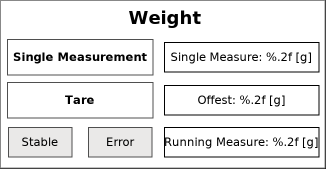
VISUALIZATION vWeighing  // 326x169
VAR_INPUT
	iNameIndex : INT;
END_VAR
VAR_IN_OUT
	fbWeighing : FB_WeighingOversampling;
END_VAR
    Rectangle (0,0 326x169)
    Rectangle (8,127 64x30), "Stable", colour toggle: fbWeighing.fbTON_ForceStable.Q
    Rectangle (114,3 102x30), "Weight", text list: 'tlDevices', text index: iNameIndex
    Rectangle (7,39 146x36), "Single Measurement"
        OnMouseDown: execute { fbWeighing.stSettings.bManualSingleMeasureRequest :=TRUE; }
    Rectangle (7,82 146x36), "Tare"
        OnMouseDown: execute { fbWeighing.stSettings.bTareRequest :=TRUE; }
    Rectangle (164,85 155x30), "Offest: %.2f [g]", text variable: fbWeighing.rZeroValue
    Rectangle (164,127 155x30), "Running Measure: %.2f [g]", text variable: fbWeighing.rRunningMeasure
    Rectangle (164,42 155x30), "Single Measure: %.2f [g]", text variable: fbWeighing.rSingleMessResult
    Rectangle (88,127 64x30), "Error", colour toggle: fbWeighing.bMeasurementError
END_VISUALIZATION

(* stored: Version 1.1.0.1, ProductVersion 3.1.4024.15
   Visu vWeighing: Id {8b33d426-e4a2-412e-aa0c-a2a04b4fed79} *)
